Staubli VAL3: setInstr.pgx

public program setInstr(InstrItem& x_iInstr[], num x_nIndex, bool x_bType)
  local string l_sInstruction
  local num i
begin
  // get the instruction and fill as an array
  if x_nIndex>=0
    // save the data
    if x_bType
      // take gun ON
      //resize(saveData:tData[x_nIndex].iActionON,1,size(x_iInstr))
      for i=0 to size(x_iInstr)-1
        saveData:tData[x_nIndex].iActionON[i]=x_iInstr[i]
      endFor
    else
      // take gun OFF
      //resize(saveData:tData[x_nIndex].iActionOFF,1,size(x_iInstr))
      for i=0 to size(x_iInstr)-1
        saveData:tData[x_nIndex].iActionOFF[i]=x_iInstr[i]
      endFor
    endIf
  endIf
end
